KUKA KRL program: chk_w8_wechs_ok.src

&ACCESS RVO20
&COMMENT Tool Change
DEF chk_w8_wechs_ok( )

; VERIFICAÇÃO DE FERRAMENTA: TOOL CHANGE


$TIMER[10] = 0
$TIMER_STOP[10] = FALSE

wait for (($IN[585] OR (NOT($IN[585]) AND ($IN[3320]))) AND (($IN[577]) OR (NOT ($IN[577]) AND ($IN[3320]))) and ( $in[161]) and ($in[169]) and (($in[177]) OR (NOT ($in[177]) and $in[3320])) and ($in[185]) and ($in[193]) and ($in[201]) and ($in[209]) AND (NOT $in[219]))

$TIMER_STOP[10] = TRUE
$TIMER[10] = 0

;//---- End -------
;Diag_Appl(#Off,5)
END
